// TIA Portal project "Project1978_clear" (V16)

(* hardware
DEVICE "S7-1200 station_1"  S7-1200 Station
   slot 0: "Rack_0"  S7-1200 Rack  Rack  V1.0
   slot 1: "PLC_1"  CPU 1214C DC/DC/DC  6ES7 214-1AG40-0XB0  V4.4
   slot 2: "DI 16x24VDC_1"  6ES7 221-1BH32-0XB0  V2.0
   slot 3: "DI 8/DQ 8x24VDC_1"  6ES7 223-1BH32-0XB0  V2.0
*)

// ===== PLC "PLC_1"  CPU 1214C DC/DC/DC =====

VAR_GLOBAL   // PLC tag table "Default tag table"
   "A11DIa_0" AT %I0.0 : Bool;
   "A11DIa_1" AT %I0.1 : Bool;
   "A11DIa_2" AT %I0.2 : Bool;
   "A11DIa_3" AT %I0.3 : Bool;
   "A11DIa_4" AT %I0.4 : Bool;
   "A11DIa_5" AT %I0.5 : Bool;
   "A11DIa_6" AT %I0.6 : Bool;
   "A11DIa_7" AT %I0.7 : Bool;
   "A11DIb_0" AT %I1.0 : Bool;
   "A11DIb_1" AT %I1.1 : Bool;
   "A11DIb_2" AT %I1.2 : Bool;
   "A11DIb_3" AT %I1.3 : Bool;
   "A11DIb_4" AT %I1.4 : Bool;
   "A11DIb_5" AT %I1.5 : Bool;
   "A11DQa_0" AT %Q0.0 : Bool;
   "A11DQa_1" AT %Q0.1 : Bool;
   "A11DQa_2" AT %Q0.2 : Bool;
   "A11DQa_3" AT %Q0.3 : Bool;
   "A11DQa_4" AT %Q0.4 : Bool;
   "A11DQa_5" AT %Q0.5 : Bool;
   "A11DQa_6" AT %Q0.6 : Bool;
   "A11DQa_7" AT %Q0.7 : Bool;
   "A11DQb_0" AT %Q1.0 : Bool;
   "A11DQb_1" AT %Q1.1 : Bool;
   "A12DIa_0" AT %I8.0 : Bool;
   "A12DIa_1" AT %I8.1 : Bool;
   "A12DIa_2" AT %I8.2 : Bool;
   "A12DIa_3" AT %I8.3 : Bool;
   "A12DIa_4" AT %I8.4 : Bool;
   "A12DIa_5" AT %I8.5 : Bool;
   "A12DIa_6" AT %I8.6 : Bool;
   "A12DIa_7" AT %I8.7 : Bool;
   "A12DIb_0" AT %I9.0 : Bool;
   "A12DIb_1" AT %I9.1 : Bool;
   "A12DIb_2" AT %I9.2 : Bool;
   "A12DIb_3" AT %I9.3 : Bool;
   "A12DIb_4" AT %I9.4 : Bool;
   "A12DIb_5" AT %I9.5 : Bool;
   "A12DIb_6" AT %I9.6 : Bool;
   "A12DIb_7" AT %I9.7 : Bool;
   "A13DIa_0" AT %I12.0 : Bool;
   "A13DIa_1" AT %I12.1 : Bool;
   "A13DIa_2" AT %I12.2 : Bool;
   "A13DIa_3" AT %I12.3 : Bool;
   "A13DIa_4" AT %I12.4 : Bool;
   "A13DIa_5" AT %I12.5 : Bool;
   "A13DIa_6" AT %I12.6 : Bool;
   "A13DIa_7" AT %I12.7 : Bool;
   "A13DQa_0" AT %Q12.0 : Bool;
   "A13DQa_1" AT %Q12.1 : Bool;
   "A13DQa_2" AT %Q12.2 : Bool;
   "A13DQa_3" AT %Q12.3 : Bool;
   "A13DQa_4" AT %Q12.4 : Bool;
   "A13DQa_5" AT %Q12.5 : Bool;
   "A13DQa_6" AT %Q12.6 : Bool;
   "A13DQa_7" AT %Q12.7 : Bool;
   "o_bAlarmStatus" AT %QW2 : Word;   // Текущее состояние ошбки
   "o_bAlarmStatus(1)" AT %QW4 : Word;   // Текущее состояние ошбки
   "i_bResetFromHMI" AT %I1.6 : Bool;   // Сброс ошибок от панели оператора
   "GlobalArarm" AT %Q1.2 : Bool;   // Глобальный флаг аварий
   "i_LocalResetUZ1" AT %I1.7 : Bool;   // Отдельный сброс для блока UZ1
   "i_LocalResetUZ1(1)" AT %I2.0 : Bool;
   "i_LocalResetUZ1(2)" AT %I2.1 : Bool;
   "System_Byte" AT %MB1 : Byte;
   "FirstScan" AT %M1.0 : Bool;
   "DiagStatusUpdate" AT %M1.1 : Bool;
   "AlwaysTRUE" AT %M1.2 : Bool;
   "AlwaysFALSE" AT %M1.3 : Bool;
   "System_Byte(1)" AT %MB1 : Byte;
   "Clock_Byte" AT %MB0 : Byte;
   "Clock_10Hz" AT %M0.0 : Bool;
   "Clock_5Hz" AT %M0.1 : Bool;
   "Clock_2.5Hz" AT %M0.2 : Bool;
   "Clock_2Hz" AT %M0.3 : Bool;
   "Clock_1.25Hz" AT %M0.4 : Bool;
   "Clock_1Hz" AT %M0.5 : Bool;
   "Clock_0.625Hz" AT %M0.6 : Bool;
   "Clock_0.5Hz" AT %M0.7 : Bool;
END_VAR

DATA_BLOCK "ResetSignals"   // DB4
{ S7_Optimized_Access := 'FALSE' }
VERSION : 0.1
   VAR
      "#i_LocalResetUZ1" : Bool;   // Отдельный сброс для блока UZ1
      i_bTurnOffLightSound : Bool;   // Сигнал отключения сигнализации
   END_VAR
BEGIN
END_DATA_BLOCK

DATA_BLOCK "JournalOfAlarm"   // DB8
{ S7_Optimized_Access := 'FALSE' }
VERSION : 0.1
   VAR
      s_bEmergButIsPressedLog : Bool;
      s_bGlobalAlarmLog : Bool;
      s_bWorkPosAlarmYA1Log : Bool;
      s_bWorkPosAlarmYA2Log : Bool;
      s_bAlarmUZ1Log : Bool;
      s_bClosePosAlarmYA1Log : Bool;
      s_bClosePosAlarmYA2Log : Bool;
      s_bNoOperationAlarmUZ1Log : Bool;
   END_VAR
BEGIN
END_DATA_BLOCK

DATA_BLOCK "JournalOfEvent"   // DB9
{ S7_Optimized_Access := 'FALSE' }
VERSION : 0.1
   VAR
      s_bManualModeLog : Bool;   // Событие выбора ручного режима
      s_bAutoModeLog : Bool;   // Событие выбора автоматического режима
      s_bAutoStartYA1Log : Bool;   // Событие запуска YA1 в авто режиме
      s_bAutoStartYA2Log : Bool;   // Событие запуска YA2 в авто режиме
      s_bAutoStartUZ1Log : Bool;   // Событие запуска UZ1 в авто режиме
      s_bManualStartYA1Log : Bool;   // Событие запуска YA1 в ручном режиме
      s_bManualStartYA2Log : Bool;   // Событие запуска YA1 в ручном режиме
      s_bManualStartUZ1Log : Bool;   // Событие запуска UZ1 в ручном режиме
      s_bAutoModeIsStartLog : Bool;   // Событие запуска автоматического режима
      s_bNoPressureInSystemLog : Bool;   // Событие отсутствия давления в системе
   END_VAR
BEGIN
END_DATA_BLOCK

// folder: AUTO&M_MODE

DATA_BLOCK "FB_Mode_DB"   // DB12
{ S7_Optimized_Access := 'FALSE' }
VERSION : 0.1
// stored: InstanceOfName FB_Mode
"FB_Mode"
BEGIN
END_DATA_BLOCK

// folder: CONVERTER

DATA_BLOCK "FB_Converter_DB"   // DB6
{ S7_Optimized_Access := 'FALSE' }
VERSION : 0.1
// stored: InstanceOfName FB_Converter
"FB_Converter"
BEGIN
   i_bConverterMode := TRUE;
   TimerStartFault.ST := T#-12D_9H_8M_40S_967MS;
   TimerStartFault.PT := T#10S;
   t_HoldForReset.ST := T#-12D_9H_8M_19S_256MS;
   t_HoldForReset.PT := T#2S;
END_DATA_BLOCK

// folder: CYLINDRES

DATA_BLOCK "FB_AlgoAutomodeCylinder_DB"   // DB1
{ S7_Optimized_Access := 'FALSE' }
VERSION : 0.1
// stored: InstanceOfName FB_AlgoAutomodeCylinder
"FB_AlgoAutomodeCylinder"
BEGIN
   i_tHoldingPusher := T#0MS;
   timeForHoldingBoxes := T#3S;
   timeForActivationPusher := T#500MS;
   timeForPreventAdhesion := T#300MS;
   o_wStatusOnFooterHMI := 16#0003;
   o_wBoxOneOnPusher := 16#0001;
   counterForStopper := 5;
   counterForPusher := 1;
   timerForPusher.ST := T#-12D_9H_37M_56S_958MS;
   timerForBoxesOnTheTable.ST := T#-12D_9H_37M_56S_958MS;
   timerForBoxesOnTheTable.PT := T#3S;
   s_bStartAuto := FALSE;
   trigBoxOneHave.CLK := TRUE;
   s_bBoxOneHaveOnTable := TRUE;
   timerForActivationPusher.ST := T#-12D_9H_37M_58S_497MS;
   timerForActivationPusher.PT := T#500MS;
   timHoldCabReset.ST := T#-12D_9H_8M_19S_255MS;
   timHoldCabReset.PT := T#3S;
   counterForStopperExtraBox := 11;
   timerAdhesion.ST := T#-12D_9H_38M_1S_127MS;
   timerAdhesion.PT := T#300MS;
END_DATA_BLOCK

DATA_BLOCK "FB_CallCylinder_DB"   // DB13
{ S7_Optimized_Access := 'FALSE' }
VERSION : 0.1
// stored: InstanceOfName FB_CallCylinder
"FB_CallCylinder"
BEGIN
   i_LocalResetYA1 := TRUE;
   i_LocalResetYA2 := TRUE;
   Pusher.i_tTimeForOpenAndClose := T#5S;
   Pusher.i_bCylinder_StartPos := TRUE;
   Pusher.i_bCylinderMode := TRUE;
   Pusher.i_b_ResetSignal := TRUE;
   Pusher.o_wStatusCylinder := 16#0001;
   Pusher.Timer_SensOpenDelay.ST := T#-12D_9H_37M_56S_962MS;
   Pusher.Timer_SensOpenDelay.PT := T#20MS;
   Pusher.Timer_SensCloseDelay.ST := T#-12D_9H_37M_55S_880MS;
   Pusher.Timer_SensCloseDelay.PT := T#20MS;
   Pusher.Timer_SensCloseDelay.IN := TRUE;
   Pusher.Timer_ClosePositionAlarm.ST := T#-12D_9H_37M_56S_954MS;
   Pusher.Timer_ClosePositionAlarm.PT := T#5S;
   Pusher.Timer_OpenPositionAlarm.ST := T#-12D_9H_37M_57S_990MS;
   Pusher.Timer_OpenPositionAlarm.PT := T#5S;
   Pusher.o_bIsStatusClosed := TRUE;
   Stopper.i_tTimeForOpenAndClose := T#2S;
   Stopper.i_bCylinder_StartPos := TRUE;
   Stopper.i_bCylinderMode := TRUE;
   Stopper.i_b_ResetSignal := TRUE;
   Stopper.o_wStatusCylinder := 16#0001;
   Stopper.Timer_SensOpenDelay.ST := T#-12D_9H_38M_962MS;
   Stopper.Timer_SensOpenDelay.PT := T#20MS;
   Stopper.Timer_SensCloseDelay.ST := T#-12D_9H_38M_611MS;
   Stopper.Timer_SensCloseDelay.PT := T#20MS;
   Stopper.Timer_SensCloseDelay.IN := TRUE;
   Stopper.Timer_ClosePositionAlarm.ST := T#-12D_9H_38M_819MS;
   Stopper.Timer_ClosePositionAlarm.PT := T#2S;
   Stopper.Timer_OpenPositionAlarm.ST := T#-12D_9H_38M_1S_123MS;
   Stopper.Timer_OpenPositionAlarm.PT := T#2S;
   Stopper.o_bIsStatusClosed := TRUE;
   ControllCyllinder.i_tHoldingPusher := T#4S;
   ControllCyllinder.i_iQuantityOfBoxes := 4;
   ControllCyllinder.timeForHoldingBoxes := T#3S;
   ControllCyllinder.s_bStartAuto := TRUE;
END_DATA_BLOCK

// folder: DI_DQ_FILLING

DATA_BLOCK "DI"   // DB2
{ S7_Optimized_Access := 'FALSE' }
VERSION : 0.1
   VAR
      i_bConveyor_UZ1_Operation : Bool;
      i_bConveyor_UZ1_Fault : Bool;
      i_bCylinder_YA1_1_StartPos : Bool;
      i_bCylinder_YA1_1_EndPos : Bool;
      i_bCylinder_YA1_2_StartPos : Bool;
      i_bCylinder_YA1_2_EndPos : Bool;
      i_bCylinder_YA2_StartPos : Bool;
      i_bCylinder_YA2_EndPos : Bool;
      i_bSensor_BL1_1_Activated : Bool;
      i_bSensor_BL1_2_Activated : Bool;
      i_bSensor_BL2_1_Activated : Bool;
      i_bSensor_BL2_2_Activated : Bool;
      i_bSensor_BL2_3_Activated : Bool;
      i_bSensor_BL2_4_Activated : Bool;
      i_bNo_Emergency_Stop_CabinetButton : Bool;
      i_bStart_CabinetButton : Bool;
      i_bStop_CabinetButton : Bool;
      i_bReset_CabinetButton : Bool;
      i_bAuto_Mode_Enabled : Bool;
      i_bStart_OperatorPanel_KP1 : Bool;
      i_bStop_OperatorPanel_KP1 : Bool;
      i_bEmergency_Stop_OperatorPanel_KP2 : Bool;
      i_bPressure_Present_PS_Relay : Bool;
   END_VAR
BEGIN
END_DATA_BLOCK

DATA_BLOCK "DQ"   // DB3
{ S7_Optimized_Access := 'FALSE' }
VERSION : 0.1
   VAR
      q_bConveyor_Start : Bool;
      q_bConveyor_Fault_Reset : Bool;
      q_bGate_Cylinder_YA1_1_Start : Bool;
      q_bGate_Cylinder_YA1_2_Start : Bool;
      q_bPusher_Cylinder_YA2_Start : Bool;
      q_bFeeder_Conveyor_Stop_Signal : Bool;
      q_bControl_BPV1 : Bool;
      q_bEmergency_LightSound_Alert : Bool;
      q_bSignallTo1C : Bool;
   END_VAR
BEGIN
END_DATA_BLOCK

// folder: DI_DQ_FILLING/ProcessInput

DATA_BLOCK "FilterInput_DB"   // DB16
{ S7_Optimized_Access := 'FALSE' }
VERSION : 0.1
// stored: InstanceOfName CallFilterInput
"CallFilterInput"
BEGIN
END_DATA_BLOCK

// folder: Modbus_TCP

DATA_BLOCK "MB_Table"   // DB1700
{ S7_Optimized_Access := 'FALSE' }
VERSION : 0.1
   VAR
      Data_Exchange : Array[0..100] of Int;
   END_VAR
BEGIN
   Data_Exchange[30] := 30;
   Data_Exchange[31] := 31;
   Data_Exchange[32] := 32;
   Data_Exchange[33] := 33;
   Data_Exchange[34] := 34;
   Data_Exchange[35] := 35;
   Data_Exchange[36] := 36;
   Data_Exchange[37] := 37;
   Data_Exchange[38] := 38;
   Data_Exchange[39] := 39;
   Data_Exchange[40] := 40;
   Data_Exchange[41] := 41;
   Data_Exchange[42] := 42;
   Data_Exchange[43] := 43;
   Data_Exchange[44] := 44;
   Data_Exchange[45] := 45;
   Data_Exchange[46] := 46;
   Data_Exchange[47] := 47;
   Data_Exchange[48] := 48;
   Data_Exchange[49] := 49;
   Data_Exchange[50] := 50;
   Data_Exchange[1] := 2;
END_DATA_BLOCK

DATA_BLOCK "ModbusTCP_DB"   // DB1701
{ S7_Optimized_Access := 'TRUE' }
VERSION : 0.1
// stored: InstanceOfName ModbusTCP
"ModbusTCP"
BEGIN
END_DATA_BLOCK

// folder: SENSORS

DATA_BLOCK "FB_CallSensor_DB"   // DB14
{ S7_Optimized_Access := 'FALSE' }
VERSION : 0.1
// stored: InstanceOfName FB_CallSensor
"FB_CallSensor"
BEGIN
   i_tDebounceTime := T#25MS;
   i_tUndebounceTime := T#10MS;
   Break.i_tDebounceTime := T#25MS;
   Break.i_tUndebounceTime := T#10MS;
   Break.tDebounceTimer.ST := T#-12D_9H_2M_33S_795MS;
   Break.tDebounceTimer.PT := T#25MS;
   Break.tUndebounceTimer.ST := T#-12D_9H_2M_33S_498MS;
   Break.tUndebounceTimer.PT := T#25MS;
   Break.tUndebounceTimer.IN := TRUE;
   Stopper.i_tDebounceTime := T#25MS;
   Stopper.i_tUndebounceTime := T#10MS;
   Stopper.tDebounceTimer.ST := T#-12D_9H_2M_43S_751MS;
   Stopper.tDebounceTimer.PT := T#25MS;
   Stopper.tUndebounceTimer.ST := T#-12D_9H_2M_37S_160MS;
   Stopper.tUndebounceTimer.PT := T#25MS;
   Stopper.tUndebounceTimer.IN := TRUE;
   "Counter".i_tDebounceTime := T#25MS;
   "Counter".i_tUndebounceTime := T#10MS;
   "Counter".tDebounceTimer.ST := T#-12D_9H_2M_34S_699MS;
   "Counter".tDebounceTimer.PT := T#25MS;
   "Counter".tUndebounceTimer.ST := T#-12D_9H_2M_34S_408MS;
   "Counter".tUndebounceTimer.PT := T#25MS;
   "Counter".tUndebounceTimer.IN := TRUE;
   CheckOnTable.i_tDebounceTime := T#25MS;
   CheckOnTable.i_tUndebounceTime := T#10MS;
   CheckOnTable.tDebounceTimer.ST := T#-12D_9H_37M_58S_309MS;
   CheckOnTable.tDebounceTimer.PT := T#25MS;
   CheckOnTable.tUndebounceTimer.ST := T#-12D_9H_37M_57S_479MS;
   CheckOnTable.tUndebounceTimer.PT := T#25MS;
   CheckOnTable.tUndebounceTimer.IN := TRUE;
END_DATA_BLOCK

// folder: System blocks/Program resources

DATA_BLOCK "Server1"   // DB5
{ S7_Optimized_Access := 'TRUE' }
AUTHOR : SIMATIC
FAMILY : MC7Plus
NAME : TC_IP_v4
VERSION : 1.0
// stored: InstanceOfName TCON_IP_v4
"TCON_IP_v4"
BEGIN
   ID := 2;
   InterfaceId := 64;
   LocalPort := 2000;
END_DATA_BLOCK

// folder: (top level)

ORGANIZATION_BLOCK "Main"   // OB1, SCL, ProgramCycle
TITLE = "Main Program Sweep (Cycle)"
{ S7_Optimized_Access := 'TRUE' }
VERSION : 0.1
   VAR_INPUT
      Initial_Call : Bool;   // Initial call of this OB
      Remanence : Bool;   // =True, if remanent data are available
   END_VAR
BEGIN
   // Инициализация Input адрессных переменных
   "IN"();

   // Инициализация кнопок шкафа
   "FilterInput_DB"();

   "ModbusTCP_DB"();

   //Инициализация режима работы
   "FB_Mode_DB"(ModeFromCabinet := "FilterInput_DB".FB_Auto_Mode_Enabled.q_FilterSignal,
                AutoStatusMode := "FB_Converter_DB".AutoStatusMode);

   // Инициализация датчиков
   "FB_CallSensor_DB"();

   // Инициализация ПЧ
   "FB_Converter_DB"(i_bExternalBlock:= NOT "FilterInput_DB".FB_No_Emergency_Stop_CabinetButton.q_FilterSignal OR "FilterInput_DB".FB_EmergencyStopOperatop.q_FilterSignal, //mb not for StopOperatop
                     i_bConveyor_UZ1_Operation := "DI".i_bConveyor_UZ1_Operation,
                     i_bConveyor_UZ1_Fault := "DI".i_bConveyor_UZ1_Fault,
                     i_bConverterMode := "FB_Mode_DB".TotalCurrentMode,
                     i_b_ResetSignal := "FilterInput_DB".FB_ResetCabinet.q_FilterSignal OR "i_bResetFromHMI" OR "ResetSignals"."#i_LocalResetUZ1",
                     i_bStop := "FilterInput_DB".FB_StopCabinet.q_FilterSignal OR "FilterInput_DB".FB_StopOperator.q_FilterSignal,
                     i_bStart :=  "FilterInput_DB".FB_StartCabinet.q_FilterSignal OR "FilterInput_DB".FB_StartOperator.q_FilterSignal,
                     i_bStartFromAuto := "FB_AlgoAutomodeCylinder_DB".o_bSignall_From_CtrlBlockToConveyor,
                     o_qConveyor_Start => "DQ".q_bConveyor_Start,
                     o_bConveyor_Fault_Reset => "DQ".q_bConveyor_Fault_Reset);

   "FB_AlgoAutomodeCylinder_DB"(i_bSensStopper:="FB_CallSensor_DB".Stopper.o_bFilteredSignal,
                                i_bSensBreak:="FB_CallSensor_DB".Break.o_bFilteredSignal,
                                i_bSensCounter:="FB_CallSensor_DB".Counter.o_bFilteredSignal);

   // Инициализация цилиндров
   "FB_CallCylinder_DB"();

   // Фиксация сигнала нажатия аварийной кнопки
   "trigFNoEmergencyButton"(CLK:="FilterInput_DB".FB_No_Emergency_Stop_CabinetButton.q_FilterSignal);
   // Логирование нажатия кнопки аварии
   "JournalOfAlarm".s_bEmergButIsPressedLog := NOT "FilterInput_DB".FB_No_Emergency_Stop_CabinetButton.q_FilterSignal OR "FilterInput_DB".FB_EmergencyStopOperatop.q_FilterSignal;


   // Действие в зависимости от выбранного режима
   IF "FB_Mode_DB".TotalCurrentMode = 1 THEN
       "DQ".q_bFeeder_Conveyor_Stop_Signal := 0;
   ELSE
       "DQ".q_bFeeder_Conveyor_Stop_Signal := 1;
   END_IF;

   // Действие при наличии хотя бы одной аварии 
   IF "FB_Converter_DB".o_bAlarmStatus > 0 OR "FB_CallCylinder_DB".Pusher.o_bAlarmStatus > 0 OR
       "FB_CallCylinder_DB".Stopper.o_bAlarmStatus > 0 OR "trigFNoEmergencyButton".Q OR
       "FilterInput_DB".FB_No_Emergency_Stop_CabinetButton.q_FilterSignal = 0 OR
        "FilterInput_DB".FB_EmergencyStopOperatop.q_FilterSignal THEN
       "GlobalArarm" := 1;
       "DQ".q_bFeeder_Conveyor_Stop_Signal := 1;
       "DQ".q_bControl_BPV1 := 0;
       "JournalOfAlarm".s_bGlobalAlarmLog := 1;
       IF NOT "ResetSignals".i_bTurnOffLightSound THEN
           "DQ".q_bEmergency_LightSound_Alert := 1;
       ELSE
           "DQ".q_bEmergency_LightSound_Alert := 0;
       END_IF;
   END_IF;

   // Взвод флага отключения сигнализации
   IF "FB_AlgoAutomodeCylinder_DB".trigRStopCabinet.Q THEN
       "ResetSignals".i_bTurnOffLightSound := 1;
   END_IF;

   // Действие при кнопке сброса от HMI или шкафа
   IF "i_bResetFromHMI" OR "FilterInput_DB".FB_ResetCabinet.q_FilterSignal THEN
       "GlobalArarm" := 0;
       "DQ".q_bEmergency_LightSound_Alert := 0;
       "DQ".q_bFeeder_Conveyor_Stop_Signal := 0;
       "DQ".q_bControl_BPV1 := 1;
       "ResetSignals".i_bTurnOffLightSound := 0;
       "JournalOfAlarm".s_bEmergButIsPressedLog := 0;
       "JournalOfAlarm".s_bGlobalAlarmLog := 0;
   END_IF;
   //"FB_CallCylinder_DB".i_LocalResetYA1 := 0;
   //"FB_CallCylinder_DB".i_LocalResetYA2 := 0;
   //"ResetSignals"."#i_LocalResetUZ1" := 0;
   // Инициализация Output адрессных переменных
   "OUT"();
END_ORGANIZATION_BLOCK

// folder: AUTO&M_MODE

FUNCTION_BLOCK "FB_Mode"   // FB10, SCL
{ S7_Optimized_Access := 'FALSE' }
VERSION : 0.1
   VAR_INPUT
      ModeFromCabinet : Bool;   // Значение от шкафа
      AutoStatusMode : Bool;   // Статус режима сейчас
   END_VAR
   VAR_OUTPUT
      TotalCurrentMode : Bool;   // Итоговый режим
   END_VAR
   VAR
      ManualValue : Bool := false;   // Используется для запуска ручного
      AutoValue : Bool := true;   // Используется для запуска авто
   END_VAR
BEGIN
   IF NOT #ModeFromCabinet THEN
       #TotalCurrentMode := 0;
       "JournalOfEvent".s_bManualModeLog := 1;
       "JournalOfEvent".s_bAutoModeLog := 0;
   END_IF;

   IF #ModeFromCabinet THEN
       #TotalCurrentMode := 1;
       "JournalOfEvent".s_bManualModeLog := 0;
       "JournalOfEvent".s_bAutoModeLog := 1;
   END_IF;
END_FUNCTION_BLOCK

// folder: CONVERTER

FUNCTION_BLOCK "FB_Converter"   // FB5, SCL
{ S7_Optimized_Access := 'FALSE' }
VERSION : 0.1
   VAR_INPUT
      i_bExternalBlock : Bool;   // Внешняя блокировка
      i_bConveyor_UZ1_Operation : Bool;   // Физ Статус работы
      i_bConveyor_UZ1_Fault : Bool;   // Физ Наличие ошибки
      i_bConverterMode : Bool;   // Режим работы от шкафа
      i_b_ResetSignal : Bool;   // Сброс от шкафа
      i_bStop : Bool;   // Стоп от кнопочного поста
      i_bStart : Bool;   // Старт от шкафа
      i_bStartManualMode_HMI : Bool;   // Старт от панели оператора
      i_bStartFromAuto : Bool;   // Старт от блока авто режима
   END_VAR
   VAR_OUTPUT
      o_bAlarmStatus : Word;   // Текущее состояние ошбки
      o_wStatusConverter : Word;   // Состояние ПЧ
      o_qConveyor_Start : Bool;   // Физ Старт
      o_bConveyor_Fault_Reset : Bool;   // Физ Сброс ошибки
      q_bAlarmForSecurityHMI : Bool;   // Битовый флаг ошибки для UZ1
   END_VAR
   VAR
      TimerDebaunceFault : TON_TIME;   // Устранение дребезга при возн аварии
      TimerStartFault : TON_TIME;   // Ошибка старта
      AutoStatusMode : Bool;   // Определение статуса работы
      ManualStatusMode : Bool;   // Статус запуска в ручном режиме
      sPositiveFrontOfTurningOn : R_TRIG;   // Опредение положительного фронта на вкл
      t_HoldForReset : TON_TIME;
      trigStartFromCab : R_TRIG;
      trigStopFromCab : R_TRIG;
      startFromCab : Bool;   // Флаг запуск/стоп от шкафа
      trigForModePos : F_TRIG;
   END_VAR
   VAR_TEMP
      PreviousStatusMode : Bool;   // Опр предыдущего статуса
   END_VAR
BEGIN
   REGION Alarm
       //Считывание статуса ошибки от конвейера
       #TimerDebaunceFault(IN := #i_bConveyor_UZ1_Fault,
                           PT := T#20ms);

       IF #TimerDebaunceFault.Q THEN
           #o_bAlarmStatus.%X0 := 1;
       END_IF;

       //Считывание статуса ошибки от конвейера при пуске 
       #TimerStartFault(IN := #o_qConveyor_Start AND NOT #i_bConveyor_UZ1_Operation,
                        PT := T#10s);

       IF #TimerStartFault.Q THEN
           #o_bAlarmStatus.%X1 := 1;
       END_IF;
       IF #i_b_ResetSignal THEN
           #o_bAlarmStatus := 0;
           "JournalOfAlarm".s_bAlarmUZ1Log := 0;
           "JournalOfAlarm".s_bNoOperationAlarmUZ1Log := 0;
           #o_bConveyor_Fault_Reset := 1;
       END_IF;

       #t_HoldForReset(IN := #o_bConveyor_Fault_Reset,
                       PT := T#2s);

       IF #t_HoldForReset.Q THEN
           #o_bConveyor_Fault_Reset := 0;
       END_IF;
   END_REGION

   REGION AutoMode
       IF #i_bConverterMode = 1 AND #i_bStartFromAuto THEN
           #AutoStatusMode := 1;
           "JournalOfEvent".s_bAutoStartUZ1Log := 1;
       END_IF;

       IF #i_bExternalBlock OR #o_bAlarmStatus > 0
           OR NOT #i_bStartFromAuto OR #i_bConverterMode = 0 THEN
           #AutoStatusMode := 0;
           "JournalOfEvent".s_bAutoStartUZ1Log := 0;
       END_IF;
   END_REGION

   REGION ManualMode
       IF #i_bConverterMode = 0 AND #i_bStartManualMode_HMI THEN
           #ManualStatusMode := 1;
           "JournalOfEvent".s_bManualStartUZ1Log := 1;
       END_IF;

       IF #i_bExternalBlock OR #o_bAlarmStatus > 0 OR NOT #i_bStartManualMode_HMI OR #i_bConverterMode = 1 OR #i_bStop THEN
           #ManualStatusMode := 0;
           "JournalOfEvent".s_bManualStartUZ1Log := 0;
       END_IF;

       IF NOT "FilterInput_DB".FB_No_Emergency_Stop_CabinetButton.q_FilterSignal
           OR "FilterInput_DB".FB_EmergencyStopOperatop.q_FilterSignal THEN
           #i_bStartManualMode_HMI := 0;
       END_IF;
   END_REGION

   #o_qConveyor_Start := #ManualStatusMode OR (#o_bAlarmStatus = 0 AND   #AutoStatusMode);

   #q_bAlarmForSecurityHMI := #o_bAlarmStatus > 0;

   #o_wStatusConverter.%X0 := #i_bConveyor_UZ1_Operation;
   #o_wStatusConverter.%X1 := #o_bAlarmStatus > 0;

   "JournalOfAlarm".s_bAlarmUZ1Log := #o_bAlarmStatus.%X0;
   "JournalOfAlarm".s_bNoOperationAlarmUZ1Log := #o_bAlarmStatus.%X1;
END_FUNCTION_BLOCK

// folder: CYLINDRES

FUNCTION_BLOCK "FB_Cylinder"   // FB1, SCL
{ S7_Optimized_Access := 'FALSE' }
VERSION : 0.1
   VAR_INPUT
      i_bStartManualMode_HMI : Bool;   // Старт от панели оператора
      i_tTimeForOpenAndClose : Time := T#10000ms;   // Время для открытия от панели
      i_bCylinder_StartPos : Bool;   // Адрессное пер закрытой позиция цилиндра
      i_bCylinderMode : Bool;   // Режим работы от шкафа
      i_bCylinder_EndPos : Bool;   // Адрессное пер открытой позиция цилиндра
      i_bExternalBlock : Bool;   // Внешняя блокировка
      i_bStart : Bool;   // Старт от блока логики
      i_bStop : Bool;   // Стоп от кнопочного поста
      i_b_ResetSignal : Bool;   // Сброс от шкафа
   END_VAR
   VAR_OUTPUT
      q_bGate_Cylinder_Start : Bool;   // Адрессная пер запуска
      o_wStatusCylinder : Word;   // Статус состояния цилиндра
      o_bAlarmStatus : Word;   // Текущее состояние ошбки
      o_bControlCylinder : Bool;   // Статус промежуточного состояния
      q_bAlarmForSecurityHMI : Bool;   // Бит аварии для панели
      o_bAlarmWorkPoslLog : Bool;   // Наличие аварии рабочего положения для логирования цилиндром
      o_bAutoStartLog : Bool;   // Логирование статуса запуска в авто режиме
      o_bManualStartLog : Bool;   // Логирование запуска в ручном режиме
      o_bAlarmClosePoslLog : Bool;   // Логирование исходного положения
   END_VAR
   VAR
      Timer_SensOpenDelay : TON_TIME;   // Таймер обработки ошибок от открытого положения
      Timer_SensCloseDelay : TON_TIME;   // Таймер обработки ошибок от закрытого положения
      Timer_ClosePositionAlarm : TON_TIME;   // Таймер опр закрытой позиции
      Timer_OpenPositionAlarm : TON_TIME;   // Таймер опр открытой позиции
      AutoStatusMode : Bool;   // Определение статуса автоматической работы
      ManualStatusMode : Bool;   // Статус запуска в ручном режиме
      sPositiveFrontOfTurningOn : R_TRIG;   // Опредение положительного фронта на вкл
      o_bIsStatusOpen : Bool;   // Проеверенный статус открытого положения
      o_bIsStatusClosed : Bool;   // Проеверенный статус закрытого положения
   END_VAR
   VAR_TEMP
      PreviousStatusMode : Bool;   // Опр предыдущего статуса
   END_VAR
BEGIN
   REGION Alarm
       #o_bControlCylinder := NOT #o_bIsStatusOpen AND NOT #o_bIsStatusClosed;

       //Статус открытого положения
       #Timer_SensOpenDelay(IN := #i_bCylinder_EndPos,
                            PT := T#20ms);
       #o_bIsStatusOpen := #Timer_SensOpenDelay.Q;

       // Блок для обработки ошибок от рабочего положения
       #Timer_OpenPositionAlarm(IN := #q_bGate_Cylinder_Start AND NOT #o_bIsStatusOpen,
                                PT := #i_tTimeForOpenAndClose);
       IF #Timer_OpenPositionAlarm.Q THEN
           #o_bAlarmStatus.%X0 := TRUE;
           #o_bAlarmWorkPoslLog := 1;
       END_IF;


       // Статус закрытого положения
       #Timer_SensCloseDelay(IN := #i_bCylinder_StartPos,
                             PT := T#20ms);
       #o_bIsStatusClosed := #Timer_SensCloseDelay.Q;

       // Блок для обработки ошибок от исходного положения
       #Timer_ClosePositionAlarm(IN := NOT #q_bGate_Cylinder_Start AND NOT #o_bIsStatusClosed,
                                 PT := #i_tTimeForOpenAndClose);
       IF #Timer_ClosePositionAlarm.Q THEN
           #o_bAlarmStatus.%X1 := TRUE;
           #o_bAlarmClosePoslLog := 1;
       END_IF;

       IF #i_b_ResetSignal THEN
           #o_bAlarmStatus := 0;
           #o_bAlarmWorkPoslLog := 0;
           #o_bAlarmClosePoslLog := 0;
       END_IF;
   END_REGION

   REGION AutoMode
       IF #i_bCylinderMode = 1 AND #i_bStart THEN
           #AutoStatusMode := 1;
           #o_bAutoStartLog := 1;
       END_IF;

       IF #i_bExternalBlock OR #i_bStop OR #i_bCylinderMode = 0 OR #i_bStart = 0 THEN
           #AutoStatusMode := 0;
           #o_bAutoStartLog := 0;
       END_IF;

       IF #i_bExternalBlock OR #o_bAlarmStatus > 0
           OR #i_bStop OR #i_bCylinderMode = 0 OR #i_bStart = 0 THEN
           #AutoStatusMode := 0;
           #o_bAutoStartLog := 0;
       END_IF;
   END_REGION

   REGION ManualMode
       IF #i_bCylinderMode = 0 AND #i_bStartManualMode_HMI THEN
           #ManualStatusMode := 1;
           #o_bManualStartLog := 1;
       END_IF;

       IF #i_bExternalBlock OR NOT #i_bStartManualMode_HMI OR #i_bCylinderMode = 1 OR #i_bStop THEN
           #ManualStatusMode := 0;
           #o_bManualStartLog := 0;
       END_IF;

       IF NOT "FilterInput_DB".FB_No_Emergency_Stop_CabinetButton.q_FilterSignal
           OR "FilterInput_DB".FB_EmergencyStopOperatop.q_FilterSignal THEN
           #i_bStartManualMode_HMI := 0;
       END_IF;
   END_REGION

   #q_bGate_Cylinder_Start := #ManualStatusMode OR (#o_bAlarmStatus = 0 AND #AutoStatusMode);

   #q_bAlarmForSecurityHMI := #o_bAlarmStatus > 0;

   #o_wStatusCylinder.%X0 := #o_bIsStatusClosed;
   #o_wStatusCylinder.%X1 := #o_bIsStatusOpen;
   #o_wStatusCylinder.%X2 := #o_bAlarmStatus > 0;
   #o_wStatusCylinder.%X3 := #q_bGate_Cylinder_Start;
END_FUNCTION_BLOCK

FUNCTION_BLOCK "FB_CallCylinder"   // FB2, SCL
{ S7_Optimized_Access := 'FALSE' }
VERSION : 0.1
   VAR_INPUT
      i_LocalResetYA1 : Bool;   // Сброс в отдельном блоке цилиндра
      i_LocalResetYA2 : Bool;   // Сброс в отдельном блоке цилиндра YA2
   END_VAR
   VAR
      Pusher : "FB_Cylinder";   // Цилиндр сдвигающий упаковки фасовщику
      Stopper : "FB_Cylinder";   // Цилиндр останавливающий упаковки
      ControllCyllinder : "FB_AlgoAutomodeCylinder";   // Алгоритм работы в автоматическом режиме
   END_VAR
BEGIN
   #Stopper(i_bExternalBlock := NOT "FilterInput_DB".FB_No_Emergency_Stop_CabinetButton.q_FilterSignal OR "FilterInput_DB".FB_EmergencyStopOperatop.q_FilterSignal, //mb not for StopOperatop
            i_bCylinder_StartPos := "DI".i_bCylinder_YA1_2_StartPos,
            i_bCylinder_EndPos := "DI".i_bCylinder_YA1_2_EndPos,
            i_bCylinderMode := "FB_Mode_DB".TotalCurrentMode,
            i_b_ResetSignal := "FilterInput_DB".FB_ResetCabinet.q_FilterSignal OR "i_bResetFromHMI" OR #i_LocalResetYA1,
            i_bStop := "FilterInput_DB".FB_StopCabinet.q_FilterSignal OR "FilterInput_DB".FB_StopOperator.q_FilterSignal,
            i_bStart := "FB_AlgoAutomodeCylinder_DB".o_bSignall_From_CtrlBlockToStopper,
            q_bGate_Cylinder_Start => "DQ".q_bGate_Cylinder_YA1_2_Start,
            o_bAlarmWorkPoslLog => "JournalOfAlarm".s_bWorkPosAlarmYA1Log,
            o_bAutoStartLog => "JournalOfEvent".s_bAutoStartYA1Log,
            o_bManualStartLog => "JournalOfEvent".s_bManualStartYA1Log,
            o_bAlarmClosePoslLog => "JournalOfAlarm".s_bClosePosAlarmYA1Log);

   #Pusher(i_bExternalBlock := NOT "FilterInput_DB".FB_No_Emergency_Stop_CabinetButton.q_FilterSignal OR "FilterInput_DB".FB_EmergencyStopOperatop.q_FilterSignal, //mb not for StopOperatop
           i_bCylinder_StartPos := "DI".i_bCylinder_YA2_StartPos,
           i_bCylinder_EndPos := "DI".i_bCylinder_YA2_EndPos,
           i_bCylinderMode := "FB_Mode_DB".TotalCurrentMode,
           i_b_ResetSignal := "FilterInput_DB".FB_ResetCabinet.q_FilterSignal OR "i_bResetFromHMI" OR #i_LocalResetYA2,
           i_bStop := "FilterInput_DB".FB_StopCabinet.q_FilterSignal OR "FilterInput_DB".FB_StopOperator.q_FilterSignal,
           i_bStart := "FB_AlgoAutomodeCylinder_DB".o_bSignall_From_CtrlBlockToPusher,
           q_bGate_Cylinder_Start => "DQ".q_bPusher_Cylinder_YA2_Start,
           o_bAlarmWorkPoslLog => "JournalOfAlarm".s_bWorkPosAlarmYA2Log,
           o_bAutoStartLog => "JournalOfEvent".s_bAutoStartYA2Log,
           o_bManualStartLog => "JournalOfEvent".s_bManualStartYA2Log,
           o_bAlarmClosePoslLog => "JournalOfAlarm".s_bClosePosAlarmYA2Log);

   "DQ".q_bSignallTo1C := #Pusher.o_bAutoStartLog;
END_FUNCTION_BLOCK

FUNCTION_BLOCK "FB_AlgoAutomodeCylinder"   // FB7, SCL
{ S7_Optimized_Access := 'FALSE' }
VERSION : 0.1
   VAR_INPUT
      i_bSensStopper : Bool;   // Сигнал от датчика стоппера
      i_tHoldingPusher : Time := T#4s;   // Время удержания пушера в открытом положении
      i_iQuantityOfBoxes : Int := 4;   // Кол-во коробок на столе фасовщика
      i_bSensBreak : Bool;   // Сигнал от датчика разрыва
      i_bSensCounter : Bool;   // Сенсор подсчета упаковок
      timeForHoldingBoxes : Time := T#3s;   // Время ужержания коробок на столе после сдвигания
      timeForActivationPusher : Time;   // Время после которого сработает пушер
      timeForPreventAdhesion : Time;   // Время после которого коробки считаются разлипшимися
   END_VAR
   VAR_OUTPUT
      o_bSignall_From_CtrlBlockToStopper : Bool;   // Актвация цилиндра-стоппера
      o_wStatusOnFooterHMI : Word;   // Отображение статуса системы в футере HMI
      o_bSignall_From_CtrlBlockToPusher : Bool;   // Активация цилиндра фасовщика
      o_bSignall_From_CtrlBlockToConveyor : Bool;   // Сигнал блоку конвейера
      o_wBoxOneOnPusher : Word;   // Отображение кол ва коробок под пушером
      o_wBoxTwoOnPusher : Word;
      o_wBoxThreeOnPusher : Word;
      o_wBoxFourOnPusher : Word;
      o_wBoxOneOnTable : Word;
      o_wBoxTwoOnTable : Word;
      o_wBoxThreeOnTable : Word;
      o_wBoxFourOnTable : Word;
   END_VAR
   VAR
      counterForStopper : Int;   // Проверка слипания
      boxesOnTheTable : Bool;   // Флаг наличия коробок на столе
      counterForPusher : Int;   // Проверка наличия 4 коробок для активации цилиндра фасовщика
      timerForStopper : TON_TIME;   // Проверка на слипание
      timerForPusher : TON_TIME;   // Для запуска при 4 упаковках
      startStopper : Bool;   // Запус стоппера
      signallFromSensStopper : R_TRIG;   // Передний фронт датчика стоппера
      signallFromSensBreak : R_TRIG;   // Передний фронт датчика слипания
      startPusher : Bool;   // Запуск пушера
      timerForBoxesOnTheTable : TON_TIME;
      triggerStartCabinet : R_TRIG;
      triggerStopAndEmergCabinet : R_TRIG;
      s_bStartAuto : Bool := true;   // Включения авторежима
      trigBoxOneHave : R_TRIG;
      s_bBoxOneHaveOnTable : Bool;   // Наличие коробки один на столе
      trigBoxTwoHave : R_TRIG;
      trigBoxThreeHave : R_TRIG;
      trigBoxFourHave : R_TRIG;
      s_bBoxTwoHaveOnTable : Bool;   // Наличие коробки два на столе
      s_bBoxThreeHaveOnTable : Bool;   // Наличие коробки три на столе
      s_bBoxFourHaveOnTable : Bool;   // Наличие коробки четыре на столе
      signallFromSensStop : F_TRIG;
      signallFromSensBreaker : F_TRIG;
      signallFromSensCount : F_TRIG;
      timerForActivationPusher : TON_TIME;
      s_bBoxOneHaveOnTableToHMI : Bool;   // Отображение коробки один в HMI
      s_bBoxTwoHaveOnTableToHMI : Bool;   // Отображение коробки два в HMI
      s_bBoxThreeHaveOnTableToHMI : Bool;   // Отображение коробки два в HMI
      s_bBoxFourHaveOnTableToHMI : Bool;   // Отображение коробки два в HMI
      timHoldCabReset : TON_TIME;
      counterForStopperExtraBox : Int;   // Счетчик наличия нужного кол ва упаковок после стоппера
      signallFromSensStopperExtra : F_TRIG;
      timerAdhesion : TON_TIME;
      signallFromSensBreakExtra : F_TRIG;
      trigRStopCabinet : R_TRIG;
      stoppingAutoMode : Bool;   // Флаг процесса остановки авто режима
   END_VAR
   VAR_TEMP
      s_bAdhesion : Bool;   // Флаг наличия слипания для счетчика коробок после стоппера
   END_VAR
BEGIN
   REGION ButtonsFromHMIandCabinet
       #triggerStartCabinet(CLK := "FilterInput_DB".FB_StartCabinet.q_FilterSignal);
       IF #triggerStartCabinet.Q THEN
           #s_bStartAuto := 1;
           "JournalOfEvent".s_bAutoModeIsStartLog := 1;
       END_IF;

       #triggerStopAndEmergCabinet(CLK := "FilterInput_DB".FB_StopCabinet.q_FilterSignal OR NOT "FilterInput_DB".FB_No_Emergency_Stop_CabinetButton.q_FilterSignal OR
                                   "FilterInput_DB".FB_EmergencyStopOperatop.q_FilterSignal);
       IF #triggerStopAndEmergCabinet.Q OR "FB_Mode_DB".TotalCurrentMode = 0 OR "GlobalArarm" = 1 THEN
           #s_bStartAuto := 0;
           "JournalOfEvent".s_bAutoModeIsStartLog := 0;
       END_IF;

       #trigRStopCabinet(CLK:="FilterInput_DB".FB_StopCabinet.q_FilterSignal);

       #timHoldCabReset(IN:="FilterInput_DB".FB_ResetCabinet.q_FilterSignal,
                        PT:=T#3s);

       IF #timHoldCabReset.Q THEN
           #counterForPusher := 0;
           #counterForStopper := 0;
           #counterForStopperExtraBox := 0;

           #o_wBoxOneOnPusher.%X0 := 0;
           #o_wBoxTwoOnPusher.%X0 := 0;
           #o_wBoxThreeOnPusher.%X0 := 0;
           #o_wBoxFourOnPusher.%X0 := 0;

           #o_wBoxOneOnTable.%X1 := 0;
           #o_wBoxTwoOnTable.%X1 := 0;
           #o_wBoxThreeOnTable.%X1 := 0;
           #o_wBoxFourOnTable.%X1 := 0;
       END_IF;
   END_REGION

   REGION Stopper
       #signallFromSensStopper(CLK := #i_bSensStopper);
       #signallFromSensBreak(CLK := #i_bSensBreak);

       #signallFromSensStopperExtra(CLK := #i_bSensStopper);

       IF #signallFromSensStopper.Q THEN
           #counterForStopper := #counterForStopper + 1;
       END_IF;

       IF #signallFromSensBreak.Q AND #counterForStopper > 0 THEN
           #counterForStopper := #counterForStopper - 1;
       END_IF;

       IF (#counterForStopper = 0 AND #i_bSensStopper AND #i_bSensBreak) OR
           (#counterForPusher >= "MB_Table".Data_Exchange[1] AND #i_bSensStopper) OR
           (#i_bSensStopper AND NOT "FB_CallCylinder_DB".Pusher.i_bCylinder_StartPos) OR
           (#counterForStopperExtraBox >= "MB_Table".Data_Exchange[1] AND #i_bSensStopper) THEN
           #startStopper := 1;
       ELSE
           #startStopper := 0;
       END_IF;

       #s_bAdhesion := #counterForStopper = 0 AND #i_bSensStopper AND #i_bSensBreak;

       #timerAdhesion(IN := #s_bAdhesion AND #i_bSensBreak,
                      PT := #timeForPreventAdhesion);

       IF #timerAdhesion.Q AND #startStopper THEN
           #counterForStopperExtraBox := #counterForStopperExtraBox + 1;
           #counterForStopper := #counterForStopper + 1;
       END_IF;

       IF #signallFromSensStopperExtra.Q THEN
           #counterForStopperExtraBox := #counterForStopperExtraBox + 1;
       END_IF;

   END_REGION

   REGION Pusher
       #signallFromSensCount(CLK:=#i_bSensCounter);

       IF #signallFromSensCount.Q THEN
           #counterForPusher := #counterForPusher + 1;
       END_IF;

       #timerForActivationPusher(IN:= #counterForPusher >= "MB_Table".Data_Exchange[1] AND NOT #boxesOnTheTable,
                                 PT:= #timeForActivationPusher);

       IF #timerForActivationPusher.Q THEN
           #startPusher := 1;
       ELSE
           #startPusher := 0;
       END_IF;

       #timerForPusher(IN := "FB_CallCylinder_DB".Pusher.i_bCylinder_EndPos,
                       PT := #i_tHoldingPusher);
       IF #timerForPusher.Q THEN
           #counterForStopper := 0;
           #counterForStopperExtraBox := 0;
           #counterForPusher := 0;
           #startPusher := 0;
           #boxesOnTheTable := 1;
       END_IF;

       #timerForBoxesOnTheTable(IN := #boxesOnTheTable,
                                PT := #timeForHoldingBoxes);
       IF #timerForBoxesOnTheTable.Q THEN
           #boxesOnTheTable := 0;

           #s_bBoxOneHaveOnTable := 0;
           #s_bBoxTwoHaveOnTable := 0;
           #s_bBoxThreeHaveOnTable := 0;
           #s_bBoxFourHaveOnTable := 0;

           #s_bBoxOneHaveOnTableToHMI := 0;
           #s_bBoxTwoHaveOnTableToHMI := 0;
           #s_bBoxThreeHaveOnTableToHMI := 0;
           #s_bBoxFourHaveOnTableToHMI := 0;
       END_IF;
   END_REGION

   #o_bSignall_From_CtrlBlockToConveyor := #s_bStartAuto AND #s_bStartAuto AND "FB_Mode_DB".TotalCurrentMode;
   #o_bSignall_From_CtrlBlockToStopper := #startStopper AND #s_bStartAuto AND "FB_Mode_DB".TotalCurrentMode;
   #o_bSignall_From_CtrlBlockToPusher := #startPusher AND #s_bStartAuto AND "FB_Mode_DB".TotalCurrentMode;

   REGION BoxOnPusher
       IF #counterForPusher = 1 THEN
           #o_wBoxOneOnPusher.%X0 := 1;
       END_IF;
       IF #counterForPusher = 2 THEN
           #o_wBoxTwoOnPusher.%X0 := 1;
       END_IF;
       IF #counterForPusher = 3 THEN
           #o_wBoxThreeOnPusher.%X0 := 1;
       END_IF;
       IF #counterForPusher = 4 THEN
           #o_wBoxFourOnPusher.%X0 := 1;
       END_IF;
       IF #counterForPusher = 0 OR "FB_CallCylinder_DB".Pusher.i_bCylinder_EndPos THEN
           #o_wBoxOneOnPusher.%X0 := 0;
           #o_wBoxTwoOnPusher.%X0 := 0;
           #o_wBoxThreeOnPusher.%X0 := 0;
           #o_wBoxFourOnPusher.%X0 := 0;
       END_IF;

       #o_wBoxOneOnPusher.%X1 := #o_bSignall_From_CtrlBlockToPusher;
       #o_wBoxTwoOnPusher.%X1 := #o_bSignall_From_CtrlBlockToPusher;
       #o_wBoxThreeOnPusher.%X1 := #o_bSignall_From_CtrlBlockToPusher;
       #o_wBoxFourOnPusher.%X1 := #o_bSignall_From_CtrlBlockToPusher;
   END_REGION

   REGION FlagBoxOnTable
   #trigBoxOneHave(CLK:=#o_wBoxOneOnPusher.%X0);
   IF #trigBoxOneHave.Q THEN
       #s_bBoxOneHaveOnTable := 1;
   END_IF;
   #trigBoxTwoHave(CLK:=#o_wBoxTwoOnPusher.%X0);
   IF #trigBoxTwoHave.Q THEN
       #s_bBoxTwoHaveOnTable := 1;
   END_IF;
   #trigBoxThreeHave(CLK:=#o_wBoxThreeOnPusher.%X0);
   IF #trigBoxThreeHave.Q THEN
       #s_bBoxThreeHaveOnTable := 1;
   END_IF;
   #trigBoxFourHave(CLK:=#o_wBoxFourOnPusher.%X0);
   IF #trigBoxFourHave.Q THEN
       #s_bBoxFourHaveOnTable := 1;
   END_IF;

   IF #s_bBoxOneHaveOnTable AND "FB_CallCylinder_DB".Pusher.i_bCylinder_EndPos THEN
       #s_bBoxOneHaveOnTableToHMI := 1;
   END_IF;
   IF #s_bBoxTwoHaveOnTable AND "FB_CallCylinder_DB".Pusher.i_bCylinder_EndPos THEN
       #s_bBoxTwoHaveOnTableToHMI := 1;
   END_IF;
   IF #s_bBoxThreeHaveOnTable AND "FB_CallCylinder_DB".Pusher.i_bCylinder_EndPos THEN
       #s_bBoxThreeHaveOnTableToHMI := 1;
   END_IF;
   IF #s_bBoxFourHaveOnTable AND "FB_CallCylinder_DB".Pusher.i_bCylinder_EndPos THEN
       #s_bBoxFourHaveOnTableToHMI := 1;
   END_IF;

       #o_wBoxOneOnTable.%X0 := 0;
       #o_wBoxTwoOnTable.%X0 := 0;
       #o_wBoxThreeOnTable.%X0 := 0;
       #o_wBoxFourOnTable.%X0 := 0;

       #o_wBoxOneOnTable.%X1 := #s_bBoxOneHaveOnTableToHMI;
       #o_wBoxTwoOnTable.%X1 := #s_bBoxTwoHaveOnTableToHMI;
       #o_wBoxThreeOnTable.%X1 := #s_bBoxThreeHaveOnTableToHMI;
       #o_wBoxFourOnTable.%X1 := #s_bBoxFourHaveOnTableToHMI;
   END_REGION

   REGION StatusOnFooterHMI
       IF "FB_Mode_DB".TotalCurrentMode <> 0 OR "FB_Mode_DB".TotalCurrentMode <> 0 THEN
           #o_wStatusOnFooterHMI := 0;
       END_IF;
       IF "FB_Mode_DB".TotalCurrentMode = 0 THEN
           #o_wStatusOnFooterHMI := 1;
       END_IF;
       IF "FB_Mode_DB".TotalCurrentMode = 0 AND ("FB_Converter_DB".ManualStatusMode OR
           "FB_CallCylinder_DB".Pusher.ManualStatusMode OR "FB_CallCylinder_DB".Stopper.ManualStatusMode) THEN
           #o_wStatusOnFooterHMI := 2;
       END_IF;
       IF "FB_Mode_DB".TotalCurrentMode THEN
           #o_wStatusOnFooterHMI := 3;
       END_IF;
       IF "FB_Mode_DB".TotalCurrentMode AND #s_bStartAuto THEN
           #o_wStatusOnFooterHMI := 4;
       END_IF;
       IF "FB_Mode_DB".TotalCurrentMode AND
           "FB_Converter_DB".i_bConveyor_UZ1_Operation AND #s_bStartAuto = 0 THEN
           #o_wStatusOnFooterHMI := 5;
       END_IF;
       IF NOT "DI".i_bPressure_Present_PS_Relay THEN
           #o_wStatusOnFooterHMI := 7;
           "JournalOfEvent".s_bNoPressureInSystemLog := 1;
       ELSE
           "JournalOfEvent".s_bNoPressureInSystemLog := 0;
       END_IF;
       IF "GlobalArarm" THEN
           #o_wStatusOnFooterHMI := 6;
       END_IF;
   END_REGION
END_FUNCTION_BLOCK

// folder: DI_DQ_FILLING

FUNCTION "IN" : Void   // FC1, SCL
{ S7_Optimized_Access := 'TRUE' }
VERSION : 0.1
BEGIN
   "DI".i_bConveyor_UZ1_Operation := "A11DIa_0";
   "DI".i_bConveyor_UZ1_Fault := "A11DIa_1";
   "DI".i_bCylinder_YA1_1_StartPos := "A11DIa_2";
   "DI".i_bCylinder_YA1_1_EndPos := "A11DIa_3";
   "DI".i_bCylinder_YA1_2_StartPos := "A11DIa_4";
   "DI".i_bCylinder_YA1_2_EndPos := "A11DIa_5";
   "DI".i_bCylinder_YA2_StartPos := "A11DIa_6";
   "DI".i_bCylinder_YA2_EndPos := "A11DIa_7";
   "DI".i_bSensor_BL1_1_Activated := "A11DIb_0";
   "DI".i_bSensor_BL1_2_Activated := "A11DIb_1";
   "DI".i_bSensor_BL2_1_Activated := "A11DIb_2";
   "DI".i_bSensor_BL2_2_Activated := "A11DIb_3";
   "DI".i_bSensor_BL2_3_Activated := "A11DIb_4";
   "DI".i_bSensor_BL2_4_Activated := "A11DIb_5";
   "DI".i_bNo_Emergency_Stop_CabinetButton := "A12DIa_0";
   "DI".i_bStart_CabinetButton := "A12DIa_1";
   "DI".i_bStop_CabinetButton := "A12DIa_2";
   "DI".i_bReset_CabinetButton := "A12DIa_3";
   "DI".i_bAuto_Mode_Enabled := "A12DIa_4";
   "DI".i_bStart_OperatorPanel_KP1 := "A12DIa_5";
   "DI".i_bStop_OperatorPanel_KP1 := "A12DIa_6";
   "DI".i_bEmergency_Stop_OperatorPanel_KP2 := "A12DIa_7";
   "DI".i_bPressure_Present_PS_Relay := "A13DIa_2";
END_FUNCTION

FUNCTION "OUT" : Void   // FC2, SCL
{ S7_Optimized_Access := 'TRUE' }
VERSION : 0.1
BEGIN
   "A11DQa_0" := "DQ".q_bConveyor_Start;
   "A11DQa_1" := "DQ".q_bConveyor_Fault_Reset;
   "A11DQa_2" := "DQ".q_bGate_Cylinder_YA1_1_Start;
   "A11DQa_3" := "DQ".q_bGate_Cylinder_YA1_2_Start;
   "A11DQa_4" := "DQ".q_bPusher_Cylinder_YA2_Start;
   "A11DQa_5" := "DQ".q_bFeeder_Conveyor_Stop_Signal;
   "A11DQa_6" := "DQ".q_bEmergency_LightSound_Alert;
   "A13DQa_7" := "DQ".q_bControl_BPV1;
   "A13DQa_6" := "DQ".q_bSignallTo1C;
END_FUNCTION

// folder: DI_DQ_FILLING/ProcessInput

FUNCTION_BLOCK "FilterInput"   // FB14, SCL
{ S7_Optimized_Access := 'TRUE' }
VERSION : 0.1
   VAR_INPUT
      i_inputSignal : Bool;
   END_VAR
   VAR_OUTPUT
      q_FilterSignal : Bool;
   END_VAR
BEGIN
   IF #i_inputSignal THEN
       #q_FilterSignal := TRUE;
   ELSE
       #q_FilterSignal := FALSE;
   END_IF;
END_FUNCTION_BLOCK

FUNCTION_BLOCK "CallFilterInput"   // FB15, SCL
{ S7_Optimized_Access := 'FALSE' }
VERSION : 0.1
   VAR
      FB_ResetCabinet : "FilterInput";
      FB_StartCabinet : "FilterInput";
      FB_StopCabinet : "FilterInput";
      FB_StartOperator : "FilterInput";
      FB_StopOperator : "FilterInput";
      FB_EmergencyStopOperatop : "FilterInput";
      FB_Auto_Mode_Enabled : "FilterInput";
      FB_No_Emergency_Stop_CabinetButton : "FilterInput";
   END_VAR
BEGIN
   #FB_ResetCabinet(i_inputSignal:="DI".i_bReset_CabinetButton);

   #FB_StartCabinet(i_inputSignal:="DI".i_bStart_CabinetButton);

   #FB_StopCabinet(i_inputSignal:="DI".i_bStop_CabinetButton);

   #FB_StartOperator(i_inputSignal:="DI".i_bStart_OperatorPanel_KP1);

   #FB_StopOperator(i_inputSignal:="DI".i_bStop_OperatorPanel_KP1);

   #FB_EmergencyStopOperatop(i_inputSignal:="DI".i_bEmergency_Stop_OperatorPanel_KP2);

   #FB_No_Emergency_Stop_CabinetButton(i_inputSignal := "DI".i_bNo_Emergency_Stop_CabinetButton);

   #FB_Auto_Mode_Enabled(i_inputSignal := "DI".i_bAuto_Mode_Enabled);
END_FUNCTION_BLOCK

// folder: Modbus_TCP

FUNCTION_BLOCK "ModbusTCP"   // FB1700, LAD
{ S7_Optimized_Access := 'TRUE' }
VERSION : 0.1
   VAR
      TCON_Server_1 : TCON;
      MB_Server_1 : MB_SERVER;
      Disconnect_S1 : Bool;   // Флаг для отключения Сервера 1
      Error_Serv1 : Word;   // Последняя ошибка Сервера 1
      TON_ReConnect_S1 : TON_TIME;   // Таймер на переподключение сервера
      TDISCON_Server_1 : TDISCON;
   END_VAR
BEGIN

REGION Network 1: Настройка сети
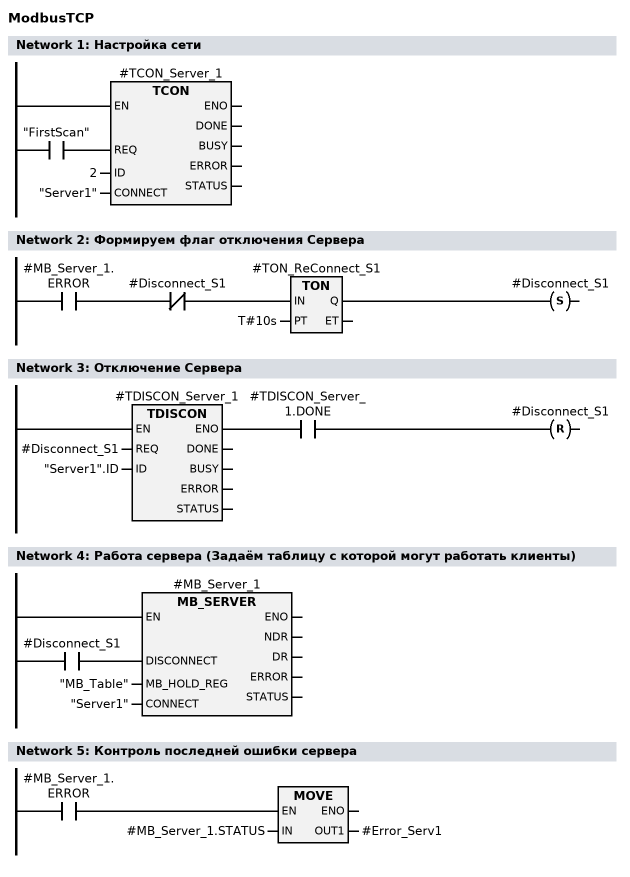
   #TCON_Server_1(REQ := "FirstScan", ID := 2, CONNECT := "Server1");   // TCON
END_REGION

REGION Network 2: Формируем флаг отключения Сервера
   #TON_ReConnect_S1(IN := #MB_Server_1.ERROR AND NOT #Disconnect_S1, PT := T#10s);   // TON
   IF #TON_ReConnect_S1.Q THEN #Disconnect_S1 := TRUE; END_IF;
END_REGION

REGION Network 3: Отключение Сервера
   // ENO of a box is taken as its EN; it also drops when the box reports an error
   #TDISCON_Server_1(REQ := #Disconnect_S1, ID := "Server1".ID);   // TDISCON
   IF #TDISCON_Server_1.DONE THEN #Disconnect_S1 := FALSE; END_IF;
END_REGION

REGION Network 4: Работа сервера (Задаём таблицу с которой могут работать клиенты)
   #MB_Server_1(DISCONNECT := #Disconnect_S1, MB_HOLD_REG := "MB_Table", CONNECT := "Server1");   // MB_SERVER
END_REGION

REGION Network 5: Контроль последней ошибки сервера
   RUNG wire#powerrail
      Contact( #MB_Server_1.ERROR )
      Move(in := #MB_Server_1.STATUS, out1 => #Error_Serv1)
   END_RUNG
   // the same network as SCL:
   IF #MB_Server_1.ERROR THEN #Error_Serv1 := #MB_Server_1.STATUS; END_IF;
END_REGION
END_FUNCTION_BLOCK

// folder: SENSORS

FUNCTION_BLOCK "FB_Sensor"   // FB3, SCL
{ S7_Optimized_Access := 'FALSE' }
VERSION : 0.1
   VAR_INPUT
      local_i_bSensor_Activated : Bool;
      i_tDebounceTime : Time;
      i_tUndebounceTime : Time := T#10ms;
   END_VAR
   VAR_OUTPUT
      o_bFilteredSignal : Bool;
   END_VAR
   VAR
      tDebounceTimer : TON_TIME;
      tActivationTimer : TON_TIME;
      tUndebounceTimer : TON_TIME;
   END_VAR
BEGIN
   #tDebounceTimer(IN := #local_i_bSensor_Activated,
                   PT := #i_tDebounceTime);

   IF #tDebounceTimer.Q THEN
       #o_bFilteredSignal := TRUE;
   END_IF;

   #tUndebounceTimer(IN := NOT #local_i_bSensor_Activated,
                     PT := #i_tDebounceTime);

   IF #tUndebounceTimer.Q THEN
       #o_bFilteredSignal := FALSE;
   END_IF;
END_FUNCTION_BLOCK

FUNCTION_BLOCK "FB_CallSensor"   // FB4, SCL
{ S7_Optimized_Access := 'FALSE' }
VERSION : 0.1
   VAR_INPUT
      i_tDebounceTime : Time := T#1ms;
      i_tUndebounceTime : Time := T#10ms;
   END_VAR
   VAR
      Break : "FB_Sensor";
      Stopper : "FB_Sensor";
      "Counter" : "FB_Sensor";
      CheckOnTable : "FB_Sensor";
   END_VAR
BEGIN
   // Датчик под отсекателем
   #Stopper(local_i_bSensor_Activated := "DI".i_bSensor_BL1_1_Activated,
            i_tDebounceTime := #i_tDebounceTime,
            i_tUndebounceTime := #i_tUndebounceTime);

   // Датчик разрыва
   #Break(local_i_bSensor_Activated := "DI".i_bSensor_BL1_2_Activated,
          i_tDebounceTime := #i_tDebounceTime,
          i_tUndebounceTime := #i_tUndebounceTime);

   // Датчик счетчика упаковок        
   #Counter(local_i_bSensor_Activated := "DI".i_bSensor_BL2_1_Activated,
            i_tDebounceTime := #i_tDebounceTime,
            i_tUndebounceTime := #i_tUndebounceTime);

   // Датчик проверки упаковок на столе
   #CheckOnTable(local_i_bSensor_Activated := "DI".i_bSensor_BL2_4_Activated,
                 i_tDebounceTime := #i_tDebounceTime,
                 i_tUndebounceTime := #i_tUndebounceTime);
END_FUNCTION_BLOCK